ABB RobotStudio station: SmartComponentSolution_20201024-152636.rsstn

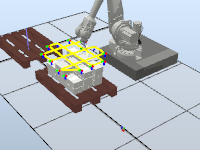
Station SmartComponentSolution (saved by RobotStudio 20.2.9116.0)
Controller IRB_4600_60kg_2.05m, task T_ROB1: task frame (RAPID world) sits at (1446.79, 1241.65, 190) mm in the station
Controller IRB_4600_60kg_2.05m
  mechanical unit ROB_1: IRB4600_60_205_C_01, 6 joints, base frame (0, -20.94, 0) mm
Layout (positions relative to the parent item):
  - IRB4600_60_205_C_01 [mechanism, from Robots\IRB4600_60_205_C_G_01.rslib] at (1446.79, 1220.71, 190) mm; joint values [-1.6147, 0.1021, 0.9055, 0, 0.5632, 1.5269] (rad or m)
  - OD1-B100H50I14-S098974 [part] at (3104.69, -456.71, 431.38) mm, rotated rx 0 ry 90 rz -90 deg
  - Box [part] at (1177.84, 251.93, 146.74) mm, rotated rx 90 ry 0 rz 0 deg
  - Euro Pallet [graphiccomponentgroup, from Equipment\Euro Pallet.rslib] at (680.82, -151.09, 0) mm
    - Body 1 [part, from Equipment\Euro Pallet.rslib] at (188.03, -194.52, 0) mm
  - SC_VaccumGripperDetector [smart component] at (1406.09, 294.35, 727.03) mm, rotated rx 180 ry 0 rz 0 deg
      signals: DO sensorSignal, DI Attached, DI Detach
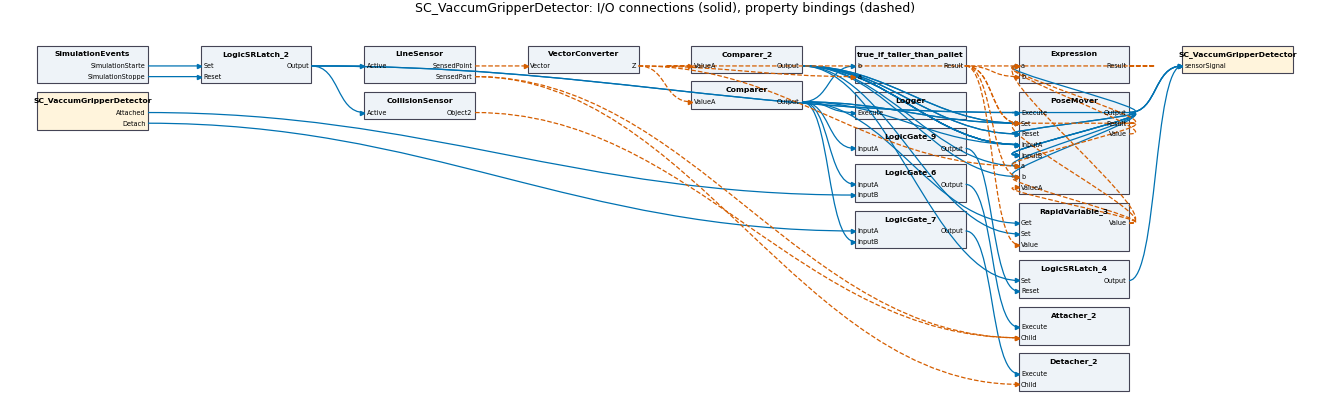
      connections:
        SimulationEvents.SimulationStarted -> LogicSRLatch_2.Set
        SimulationEvents.SimulationStopped -> LogicSRLatch_2.Reset
        LogicSRLatch_2.Output -> LineSensor.Active
        LogicSRLatch_2.Output -> PoseMover.Execute
        LogicSRLatch_2.Output -> Positioner.Execute
        Comparer.Output -> LogicSRLatch_6.Set
        LogicSRLatch_6.Output -> PoseMover_3.Execute
        LogicSRLatch_6.Output -> SC_VaccumGripperDetector.sensorSignal
        Comparer.Output -> LogicGate_6.InputA
        SC_VaccumGripperDetector.Attached -> LogicGate_6.InputB
        LogicGate_6.Output -> Attacher_2.Execute
        SC_VaccumGripperDetector.Detach -> LogicGate_7.InputA
        Comparer.Output -> LogicGate_7.InputB
        LogicGate_7.Output -> Detacher_2.Execute
        Comparer.Output -> Logger.Execute
        Comparer.Output -> true_if_taller_than_pallete.b
        Comparer_2.Output -> LogicSRLatch_4.Reset
        LogicSRLatch_4.Output -> Expression.a
        Comparer.Output -> LogicGate_8.InputA
        LogicSRLatch_4.Output -> LogicGate_8.InputB
        LogicGate_8.Output -> SC_VaccumGripperDetector.sensorSignal
        Comparer_2.Output -> Expression_3.a
        Comparer_2.Output -> LogicGate_9.InputA
        LogicSRLatch_5.Output -> LogicGate_9.InputB
        Comparer_2.Output -> LogicGate_10.InputA
        Comparer_2.Output -> LogicGate_12.InputA
        LogicGate_12.Output -> LogicSRLatch_5.Reset
        Comparer_2.Output -> LogicGate_13.InputA
        Comparer.Output -> LogicSRLatch_5.Set
        LogicSRLatch_5.Output -> Expression_4.b
        Comparer_2.Output -> LogicSRLatch_5.Reset
        Comparer_2.Output -> Expression_6.b
        Comparer_2.Output -> LogicSRLatch_7.Set
        LogicSRLatch_2.Output -> CollisionSensor.Active
        Comparer_2.Output -> LogicSRLatch_3.Set
        LogicSRLatch_3.Output -> SC_VaccumGripperDetector.sensorSignal
        Comparer_2.Output -> LogicGate_8.InputA
        LogicSRLatch_3.Output -> LogicGate_8.InputB
        LogicGate_8.Output -> LogicSRLatch_3.Reset
        Comparer_3.Output -> Expression_2.a
        Comparer.Output -> RapidVariable_3.Get
        Comparer_2.Output -> RapidVariable_3.Set
        LogicSRLatch_4.Output -> SC_VaccumGripperDetector.sensorSignal
        Comparer_2.Output -> LogicSRLatch_4.Set
        LogicGate_9.Output -> LogicSRLatch_4.Reset
        Comparer.Output -> LogicGate_9.InputA
        LineSensor.SensedPoint => VectorConverter.Vector
        VectorConverter.Z => Comparer.ValueA
        VectorConverter.Z => Expression.a
        LineSensor.SensedPart => Attacher_2.Child
        LineSensor.SensedPart => Detacher_2.Child
        Expression.Result => Comparer_2.ValueA
        VectorConverter.Z => true_if_taller_than_pallete.a
        true_if_taller_than_pallete.Result => LogicSRLatch_4.Set
        true_if_taller_than_pallete.Result => Expression.b
        true_if_taller_than_pallete.Result => Expression_3.b
        Expression_3.Result => LogicSRLatch_6.Set
        Expression_3.Result => Expression_4.a
        RapidVariable.Value => Expression.a
        true_if_taller_than_pallete.Result => RapidVariable_2.Set
        true_if_taller_than_pallete.Result => RapidVariable_3.Value
        RapidVariable_3.Value => LogicSRLatch_7.Set
        CollisionSensor.Object2 => Attacher_2.Child
        RapidVariable_3.Value => Comparer_3.ValueA
        RapidVariable_3.Value => Expression_2.b
        Expression_2.Result => Expression.a
        RapidVariable_3.Value => Expression.a
    - small_suction_gripper_2 [mechanism] at (0, 0, 0.06) mm
        TCP small_suction_gripper at (-62.96, -41.92, 61.7) mm, rotated rx 90 ry 0 rz 0 deg
        links: suction gripper-2_3
    - LineSensor [smart component, from Components\LineSensor.rslib] at (-638.5, 408.61, -364.87) mm
        properties: Start=[0.641250538776752 -0.457606 0.455378]; End=[0.641250538776752 -0.457606 1.042378]; Radius=0.001; SensedPart=Box_21; SensedPoint=[1.44807238769531 0.315089965820313 0.455770446777344]
      - _sensorPart_ [part]
    - Comparer [smart component, from Components\Comparer.rslib]
        properties: ValueA=0.455770446777344; Operator=>; ValueB=0.2
    - VectorConverter [smart component, from Components\VectorConverter.rslib]
        properties: X=1.44807238769531; Y=0.315089965820313; Z=0.455770446777344; Vector=[1.44807238769531 0.315089965820313 0.455770446777344]
    - SimulationEvents [smart component, from Components\SimulationEvents.rslib]
    - LogicSRLatch_2 [smart component, from Components\LogicSRLatch.rslib]
    - Attacher_2 [smart component, from Components\Attacher.rslib]
        properties: Parent=small_suction_gripper_2; Flange=0; Child=Box_21; Mount=false; Offset=[0 0 0]; Orientation=[0 0 0]
    - LogicGate_6 [smart component, from Components\LogicGate.rslib]
        properties: Operator=AND; Delay=0
    - Detacher_2 [smart component, from Components\Detacher.rslib]
        properties: Child=Box_21; KeepPosition=true
    - LogicGate_7 [smart component, from Components\LogicGate.rslib]
        properties: Operator=AND; Delay=0
    - Logger [smart component, from Components\Logger.rslib]
        properties: Format=Detected point; Message=Detected point; Severity=0
    - Expression [smart component, from Components\Expression.rslib]
        properties: Expression=abs(a-b) ; Result=0; a=0.455770446777344; b=0.455770446777344
    - Comparer_2 [smart component, from Components\Comparer.rslib]
        properties: ValueA=0; Operator=>; ValueB=0.01
    - true_if_taller_than_pallete [smart component, from Components\Expression.rslib]
        properties: Expression=a*b; Result=0.455770446777344; a=0.455770446777344; b=1
    - RapidVariable_3 [smart component, from Components\RapidVariable.rslib]
        properties: DataType=num; Controller=IRB_4600_60kg_2.05m; Task=T_ROB1; Module=Module1; Variable=previousBest; Value=0.455770446777344
    - CollisionSensor [smart component, from Components\CollisionSensor.rslib]
        properties: Object1=small_suction_gripper_2; Object2=(none); NearMiss=0.003; Part1=DEFAULT-32; Part2=Connector_2; CollisionType=2
    - LogicSRLatch_4 [smart component, from Components\LogicSRLatch.rslib]
    - LogicGate_9 [smart component, from Components\LogicGate.rslib]
        properties: Operator=NOT; Delay=0
  - OD1-B100H50I14-S098974_2 [part] at (1340.98, 342.45, 660.52) mm, rotated rx 0 ry -90 rz -90 deg
  - Connector_2 [part] at (1398.43, 303.95, 704.53) mm, rotated rx -90 ry 0 rz 0 deg
  - Box_3 [part] at (1185.99, -122.34, 146.74) mm, rotated rx 90 ry 0 rz 0 deg
  - Box_4 [part] at (1445.39, 246.82, 146.74) mm, rotated rx 90 ry 0 rz 0 deg
  - Box_5 [part] at (1444.81, 62.3, 146.74) mm, rotated rx 90 ry 0 rz 0.02 deg
  - Box_6 [part] at (1450.77, -121.78, 146.74) mm, rotated rx 90 ry 0 rz 0 deg
  - Box_7 [part] at (1706.66, 246.81, 146.74) mm, rotated rx 90 ry 0 rz 0 deg
  - Box_8 [part] at (1709.65, 54.45, 146.74) mm, rotated rx 90 ry 0 rz -0.01 deg
  - Box_9 [part] at (1718.44, -127.61, 146.74) mm, rotated rx 90 ry 0 rz 0 deg
  - Euro Pallet_2 [graphiccomponentgroup, from Equipment\Euro Pallet.rslib] at (-902.1, -151.09, 0) mm
    - Body 1 [part, from Equipment\Euro Pallet.rslib] at (188.03, -194.52, 0) mm
  - LogicSRLatch_7 [smart component, from Components\LogicSRLatch.rslib]
  - LogicGate_4 [smart component, from Components\LogicGate.rslib]
      properties: Operator=NOT; Delay=0
  - Base [part] at (942.52, 936.84, 0) mm
  - Box_10 [part] at (1718.44, -126.89, 251.14) mm, rotated rx 90 ry 0 rz 0 deg
  - Box_11 [part] at (1719.59, 55.71, 251.14) mm, rotated rx 90 ry 0 rz -0.03 deg
  - Box_12 [part] at (1718.45, 248.63, 251.14) mm, rotated rx 90 ry 0 rz 0 deg
  - Box_13 [part] at (1436.4, 251.82, 251.14) mm, rotated rx 90 ry 0 rz 0 deg
  - Box_14 [part] at (1172.16, 252.3, 251.14) mm, rotated rx 90 ry 0 rz 0 deg
  - Box_15 [part] at (1452.41, 56.31, 251.14) mm, rotated rx 90 ry 0 rz 0 deg
  - Box_17 [part] at (1451.15, -126.89, 251.14) mm, rotated rx 90 ry 0 rz 0 deg
  - Box_18 [part] at (1177.85, -126.84, 251.14) mm, rotated rx 90 ry 0 rz 0 deg
  - Box_19 [part] at (1451.14, -126.95, 355.53) mm, rotated rx 90 ry 0 rz 0 deg
  - Box_20 [part] at (1449.67, 54.99, 355.53) mm, rotated rx 90 ry 0 rz -0.03 deg
  - Box_21 [part] at (1451.16, 254.59, 355.53) mm, rotated rx 90 ry 0 rz 0 deg
  - Box_28 [part] at (1726.18, 254.62, 355.53) mm, rotated rx 90 ry 0 rz 0 deg
  - Box_29 [part] at (1189.3, 254.67, 355.53) mm, rotated rx 90 ry 0 rz 0 deg
  - Box_30 [part] at (1717.86, 58.35, 355.53) mm, rotated rx 90 ry 0 rz -0.02 deg
  - Frame_1 [frame] at (3169.8, -408.61, 483.89) mm
Attachment: OD1-B100H50I14-S098974_2 is attached to DEFAULT-34
Attachment: Connector_2 is attached to DEFAULT-34
Attachment: SC_VaccumGripperDetector is attached to IRB4600_60_205_C_01 / Link6
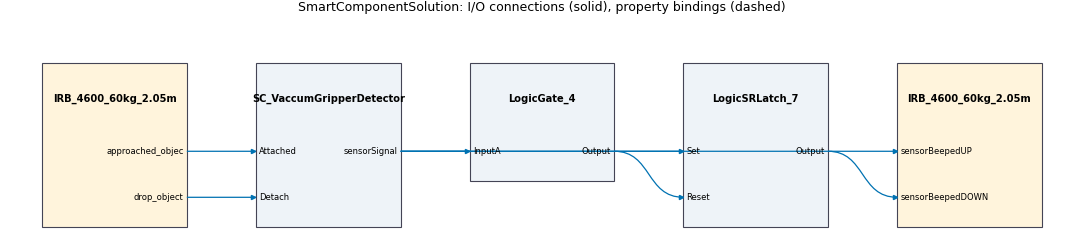
Station logic (signal -> signal, property => property):
  SC_VaccumGripperDetector.sensorSignal -> IRB_4600_60kg_2.05m.sensorBeepedUP
  SC_VaccumGripperDetector.sensorSignal -> LogicSRLatch_7.Set
  SC_VaccumGripperDetector.sensorSignal -> LogicGate_4.InputA
  LogicGate_4.Output -> LogicSRLatch_7.Reset
  LogicSRLatch_7.Output -> IRB_4600_60kg_2.05m.sensorBeepedDOWN
  IRB_4600_60kg_2.05m.approached_object -> SC_VaccumGripperDetector.Attached
  IRB_4600_60kg_2.05m.drop_object -> SC_VaccumGripperDetector.Detach
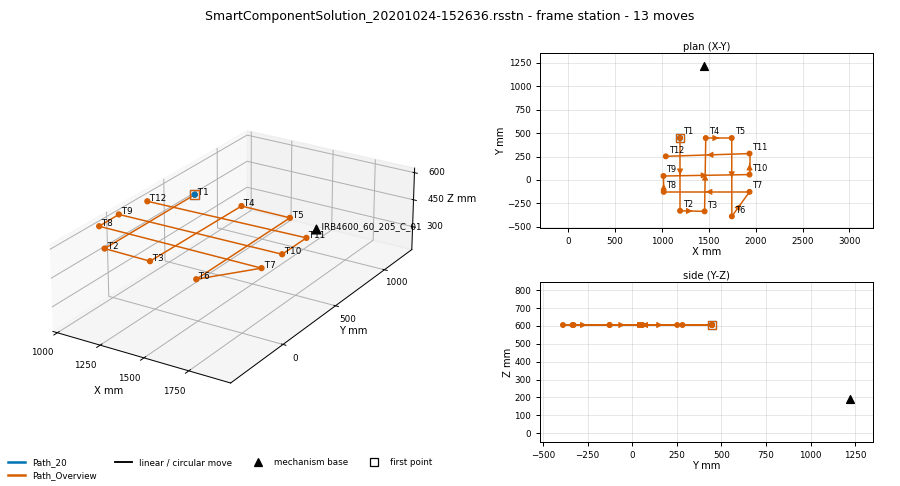
[picture p0: tool path of SmartComponentSolution_20201024-152636.rsstn in frame station, 13 of 13 moves have a stored position in this frame; points joined in program order, loops and branches not executed]
Targets, tools, work objects and paths stored in the station, written as RAPID:
! task T_ROB1
MODULE Module1
  CONST robtarget T1:=[[-252.987593195,-794.399358017,415.526565821],[0,1,0,0],[0,0,0,0],[9E+09,9E+09,9E+09,9E+09,9E+09,9E+09]];
  CONST robtarget T2:=[[-252.987593195,-1570.633594251,415.526565821],[0,1,0,0],[0,0,0,0],[9E+09,9E+09,9E+09,9E+09,9E+09,9E+09]];
  CONST robtarget T3:=[[8.712152916,-1576.575411719,415.526565821],[0,1,0,0],[0,0,0,0],[9E+09,9E+09,9E+09,9E+09,9E+09,9E+09]];
  CONST robtarget T4:=[[21.135985431,-794.399358017,415.526565821],[0,1,0,0],[0,0,0,0],[9E+09,9E+09,9E+09,9E+09,9E+09,9E+09]];
  CONST robtarget T5:=[[298.25164601,-794.399358017,415.526565821],[0,1,0,0],[0,0,0,0],[9E+09,9E+09,9E+09,9E+09,9E+09,9E+09]];
  CONST robtarget T6:=[[299.291675427,-1629.961321583,415.526565821],[0,1,0,0],[0,0,0,0],[9E+09,9E+09,9E+09,9E+09,9E+09,9E+09]];
  CONST robtarget T7:=[[488.182496173,-1368.656101944,415.526565821],[0,1,0,0],[0,0,0,0],[9E+09,9E+09,9E+09,9E+09,9E+09,9E+09]];
  CONST robtarget T8:=[[-427.404409552,-1368.656101944,415.526565821],[0,1,0,0],[0,0,0,0],[9E+09,9E+09,9E+09,9E+09,9E+09,9E+09]];
  CONST robtarget T9:=[[-430.017670434,-1199.600999294,415.526565821],[0,1,0,0],[0,0,0,0],[9E+09,9E+09,9E+09,9E+09,9E+09,9E+09]];
  CONST robtarget T10:=[[488.182496173,-1184.286468635,415.526565821],[0,1,0,0],[0,0,0,0],[9E+09,9E+09,9E+09,9E+09,9E+09,9E+09]];
  CONST robtarget T11:=[[488.182496173,-960.24487092,415.526565821],[0,1,0,0],[0,0,0,0],[9E+09,9E+09,9E+09,9E+09,9E+09,9E+09]];
  CONST robtarget T12:=[[-404.863695876,-989.636978284,415.526565821],[0,1,0,0],[0,0,0,0],[9E+09,9E+09,9E+09,9E+09,9E+09,9E+09]];
  CONST robtarget HelpPoint:=[[471.941144739,-1629.961321583,415.526565821],[0,1,0,0],[0,0,0,0],[9E+09,9E+09,9E+09,9E+09,9E+09,9E+09]];
  PROC main()
    Path_20;
  ENDPROC
  PROC Path_20()
    MoveL T1,v80,z100,small_suction_gripper\WObj:=wobj0;
  ENDPROC
  PROC Path_Overview()
    MoveL T1,v1000,z100,small_suction_gripper\WObj:=wobj0;
    MoveL T2,v1000,z100,small_suction_gripper\WObj:=wobj0;
    MoveL T3,v1000,z100,small_suction_gripper\WObj:=wobj0;
    MoveL T4,v1000,z100,small_suction_gripper\WObj:=wobj0;
    MoveL T5,v1000,z100,small_suction_gripper\WObj:=wobj0;
    MoveL T6,v1000,z100,small_suction_gripper\WObj:=wobj0;
    MoveL T7,v1000,z100,small_suction_gripper\WObj:=wobj0;
    MoveL T8,v1000,z100,small_suction_gripper\WObj:=wobj0;
    MoveL T9,v1000,z100,small_suction_gripper\WObj:=wobj0;
    MoveL T10,v1000,z100,small_suction_gripper\WObj:=wobj0;
    MoveL T11,v1000,z100,small_suction_gripper\WObj:=wobj0;
    MoveL T12,v1000,z100,small_suction_gripper\WObj:=wobj0;
  ENDPROC
ENDMODULE

! task T_ROB1
MODULE CalibData
  PERS tooldata small_suction_gripper:=[TRUE,[[-0.000055309,0.000726868,121.499905969],[1,0.000000005,0.000000013,-0.000000029]],[1,[0.443001337,-9.457000743,69.908999891],[1,0,0,0],0,0,0]];
ENDMODULE

